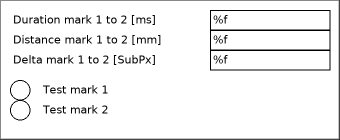
VISUALIZATION _VISU_NeutralFiberDetermine  // 340x140
VAR_IN_OUT
	mInst : FB_NeutralFibreDetermine;
END_VAR
    Rectangle (0,0 340x140)
    Rectangle (10,10 180x20), "Duration mark 1 to 2 [ms]"
    Rectangle (210,10 120x20), "%f", text variable: mInst.fL_DurationMark01to02 / 1000
    Rectangle (10,30 180x20), "Distance mark 1 to 2 [mm]"
    Rectangle (210,30 120x20), "%f", text variable: mInst.fL_LengthMark01to02
        OnMouseClick: write the text variable via Default
    Rectangle (10,50 180x20), "Delta mark 1 to 2 [SubPx]"
    Rectangle (210,50 120x20), "%f", text variable: mInst.nL_DeltaMark01to02
        OnMouseClick: write the text variable via Default
    Ellipse (10,80 20x20), tooltip "Sim VEncoder"
        tap mInst.bIKp_MarkTrigger01
    Rectangle (40,80 100x20), "Test mark 1"
    Ellipse (10,100 20x20), tooltip "Sim VEncoder"
        tap mInst.bIKp_MarkTrigger02
    Rectangle (40,100 100x20), "Test mark 2"
END_VISUALIZATION

(* stored: Version 1.1.0.1, ProductVersion 3.1.4024.11
   Visu _VISU_NeutralFiberDetermine: Id {913003fd-6449-448b-a9a2-c8c67d958e8f} *)
